Universal Robots PolyScope program: ControlSet2.urp

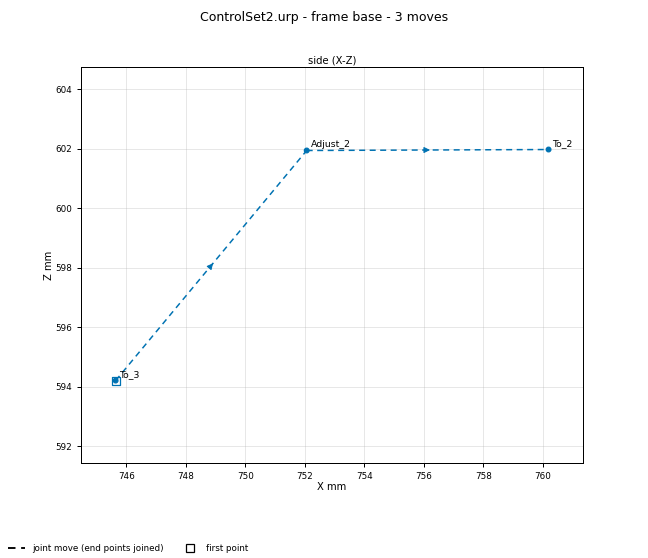
[picture p0: tool path of ControlSet2.urp in frame base, 3 of 5 moves have a stored position in this frame; points joined in program order, loops and branches not executed]
Program ControlSet2 (installation=Youssef directory=/programs/Youssef createdIn=5.9.5.1031259 lastSavedIn=5.9.5.1031259 robotSerialNumber=20215500597)
Calibrated DH parameters: a=[0.000193, -0.066673, -0.391568, -0.000012, 0.00005, 0]; d=[0.162643, -472.05677, 465.132521, 7.058239, 0.099746, 0.099582]; alpha=[1.571116, 0.00089, 0.003862, 1.569269, -1.569248, 0]; deltaTheta=[0, -1.413394, 7.628392, 0.068187, 0, -0.000001]
Robot Program (runOnlyOnce=false)
  MoveJ speed 60 deg/s, acceleration 80 deg/s^2 (useActiveTCP=true) feature=Base
    Waypoint Waypoint (Variable): variable(featureName=Control_Standby)
    Waypoint Waypoint (Variable): variable(featureName=Control_R_Strt)
    Waypoint To_3: TCP in base x=745.639 y=-17.849 z=594.209 mm, rx=-0.0636 ry=2.4703 rz=-0.2743 rad; joints [169.914, -71.977, 43.233, -100.537, -93.87, 75.587] deg; TCP offset x=0 y=0 z=191.5 mm, rx=0 ry=0 rz=0 rad
  MoveJ speed 60 deg/s, acceleration 80 deg/s^2 (useActiveTCP=true) feature=Base
    Waypoint Adjust_2: TCP in base x=752.062 y=-17.854 z=601.945 mm, rx=-0.0636 ry=2.4704 rz=-0.2743 rad; joints [170.031, -70.021, 39.176, -98.427, -93.941, 75.669] deg
    Waypoint To_2: TCP in base x=760.195 y=-17.853 z=601.978 mm, rx=-0.0636 ry=2.4703 rz=-0.2743 rad; joints [170.175, -68.462, 36.913, -97.718, -94.032, 75.776] deg
